FUNCTION_BLOCK FB_LiftA_Extended EXTENDS FB_Lift
VAR_INPUT
	i_aLayerHeights	: ARRAY[1..10] OF INT;
	i_iLayerCount: INT;
	i_eZuigerDone : eZuigerCilinderPosition;
END_VAR
VAR_OUTPUT
	o_xGoSchuif: BOOL;
	o_xGoZuiger: BOOL;
	o_xLiftDone: BOOL;
END_VAR
VAR
	LayerState: INT;
END_VAR

SUPER^();

IF i_xPalletInPosition THEN
	THIS^.MoveUpToLayer();
END_IF

METHOD MoveHome : BOOL
VAR_INPUT
END_VAR
END_METHOD

METHOD MoveUpToLayer : BOOL
VAR_INPUT
END_VAR

VAR
	CurrentLayer: INT;
END_VAR
CASE LayerState OF
	0: // Idle / Start
		CurrentLayer := 1;
	
		IF i_iLayerCount > 0 THEN
			LayerState := 1;
		END_IF
	
	
	1: // Move to current layer
		o_iTargetPos := i_aLayerHeights[CurrentLayer];
		o_xMotor := TRUE;
	
		IF i_iServoEncoder = o_iTargetPos THEN
			o_xMotor := FALSE;
			LayerState := 2;
		END_IF
	
	
	2: // Do action at layer
		o_xGoZuiger := TRUE;	// Use Zuiger to remove any layer cartons
		IF i_eZuigerDone = eZuigerCilinderPosition.Up THEN
			o_xGoSchuif := TRUE;	// Push cans onto conveyor
		END_IF
		
		IF i_xMoveUpSafe THEN
			LayerState := 3;
		END_IF
	
	3: // Advance to next layer
		CurrentLayer := CurrentLayer + 1;
	
		IF CurrentLayer > i_iLayerCount THEN
			LayerState := 4;   // all layers done
		ELSE
			LayerState := 1;   // go to next layer
		END_IF
	
	
	4: // Finished
		THIS^.MoveHome();
		// wait here

END_CASE
END_METHOD

END_FUNCTION_BLOCK

(* stored: Version 1.1.0.1
   POU FB_LiftA_Extended: Id {ae4ed0eb-eafe-4c35-b8eb-4223fd698d69}, SpecialFunc None
   Method MoveHome: Id {4513c6c0-0989-4c7f-b9dc-fd6793baeddd}
   Method MoveUpToLayer: Id {a3b1756c-3dc2-4e81-9a1c-b2a3ad14fbe2} *)
